SYSTEM sorting_by_height_basic
  (* Version 1.0, 2022-10-03, AK123957 *)
  APPLICATION sorting_by_height_basicApp
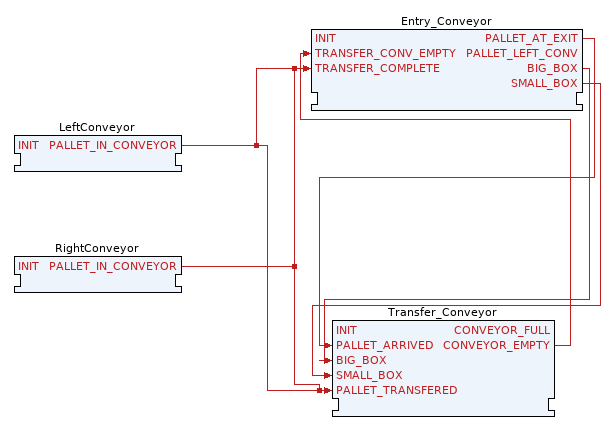
    SUBAPPLICATION Entry_Conveyor
      EVENT_INPUT
        INIT;
        TRANSFER_CONV_EMPTY;
        TRANSFER_COMPLETE;
      END_EVENT
      EVENT_OUTPUT
        PALLET_AT_EXIT;
        PALLET_LEFT_CONV;
        BIG_BOX;
        SMALL_BOX;
      END_EVENT
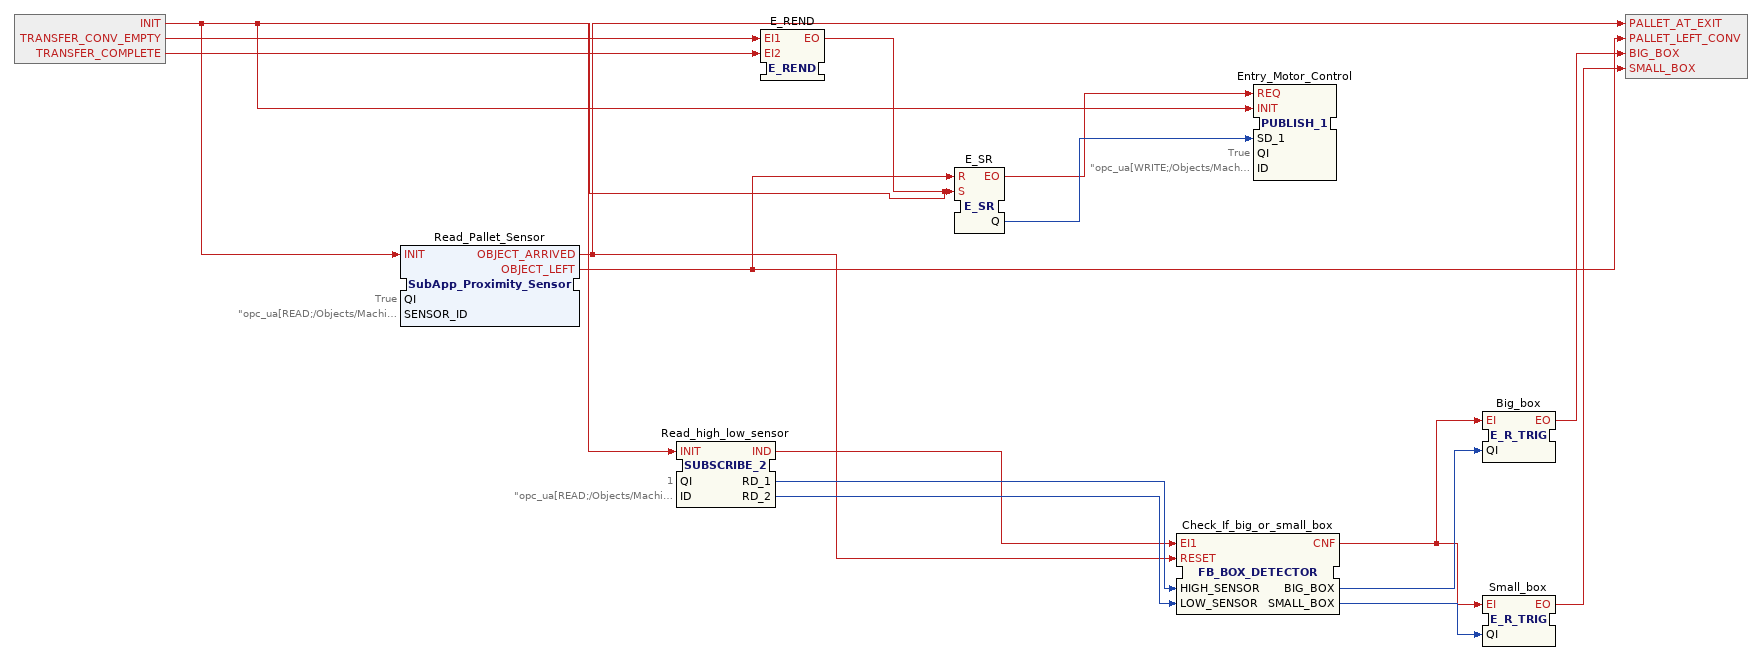
      FBS
        Entry_Motor_Control : PUBLISH_1(QI := True, ID := "opc_ua[WRITE;/Objects/Machines/EntryConveyor/FIO_oEntryMotor,1:s=FIO_oEntryMotor]");
        E_SR : E_SR;
        Check_If_big_or_small_box : FB_BOX_DETECTOR;
        Read_high_low_sensor : SUBSCRIBE_2(QI := 1, ID := "opc_ua[READ;/Objects/Machines/EntryConveyor/FIO_iHighSensor,1:s=FIO_iHighSensor;/Objects/Machines/EntryConveyor/FIO_iLowSensor,1:s=FIO_iLowSensor]");
        Big_box : E_R_TRIG;
        Small_box : E_R_TRIG;
        E_REND : E_REND;
      END_FBS
      SUBAPPS
        Read_Pallet_Sensor : SubApp_Proximity_Sensor(QI := True, SENSOR_ID := "opc_ua[READ;/Objects/Machines/EntryConveyor/FIO_iPalletSensor,1:s=FIO_iPalletSensor]");
      END_SUBAPPS
      EVENT_CONNECTIONS
        E_SR.EO TO Entry_Motor_Control.REQ;
        Read_Pallet_Sensor.OBJECT_ARRIVED TO PALLET_AT_EXIT;
        Read_Pallet_Sensor.OBJECT_LEFT TO PALLET_LEFT_CONV;
        INIT TO Read_Pallet_Sensor.INIT;
        Read_high_low_sensor.IND TO Check_If_big_or_small_box.EI1;
        Read_Pallet_Sensor.OBJECT_ARRIVED TO Check_If_big_or_small_box.RESET;
        Check_If_big_or_small_box.CNF TO Big_box.EI;
        Check_If_big_or_small_box.CNF TO Small_box.EI;
        Big_box.EO TO BIG_BOX;
        Small_box.EO TO SMALL_BOX;
        INIT TO Read_high_low_sensor.INIT;
        INIT TO Entry_Motor_Control.INIT;
        Read_Pallet_Sensor.OBJECT_LEFT TO E_SR.R;
        TRANSFER_CONV_EMPTY TO E_REND.EI1;
        TRANSFER_COMPLETE TO E_REND.EI2;
        E_REND.EO TO E_SR.S;
        INIT TO E_SR.S;
      END_CONNECTIONS
      DATA_CONNECTIONS
        E_SR.Q TO Entry_Motor_Control.SD_1;
        Read_high_low_sensor.RD_1 TO Check_If_big_or_small_box.HIGH_SENSOR;
        Read_high_low_sensor.RD_2 TO Check_If_big_or_small_box.LOW_SENSOR;
        Check_If_big_or_small_box.BIG_BOX TO Big_box.QI;
        Check_If_big_or_small_box.SMALL_BOX TO Small_box.QI;
      END_CONNECTIONS
    END_SUBAPPLICATION
    SUBAPPLICATION LeftConveyor
      EVENT_INPUT
        INIT;
      END_EVENT
      EVENT_OUTPUT
        PALLET_IN_CONVEYOR;
      END_EVENT
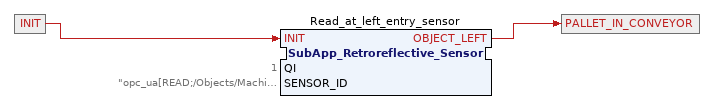
      SUBAPPS
        Read_at_left_entry_sensor : SubApp_Retroreflective_Sensor(QI := 1, SENSOR_ID := "opc_ua[READ;/Objects/Machines/LeftConveyor/FIO_iAtLeftEntry,1:s=FIO_iAtLeftEntry]");
      END_SUBAPPS
      EVENT_CONNECTIONS
        INIT TO Read_at_left_entry_sensor.INIT;
        Read_at_left_entry_sensor.OBJECT_LEFT TO PALLET_IN_CONVEYOR;
      END_CONNECTIONS
    END_SUBAPPLICATION
    SUBAPPLICATION RightConveyor
      EVENT_INPUT
        INIT;
      END_EVENT
      EVENT_OUTPUT
        PALLET_IN_CONVEYOR;
      END_EVENT
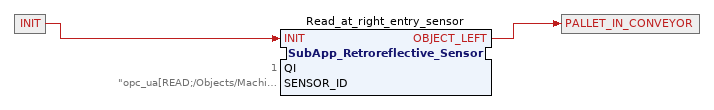
      SUBAPPS
        Read_at_right_entry_sensor : SubApp_Retroreflective_Sensor(QI := 1, SENSOR_ID := "opc_ua[READ;/Objects/Machines/RightConveyor/FIO_iAtRightEntry,1:s=FIO_iAtRightEntry]");
      END_SUBAPPS
      EVENT_CONNECTIONS
        INIT TO Read_at_right_entry_sensor.INIT;
        Read_at_right_entry_sensor.OBJECT_LEFT TO PALLET_IN_CONVEYOR;
      END_CONNECTIONS
    END_SUBAPPLICATION
    SUBAPPLICATION Transfer_Conveyor
      EVENT_INPUT
        INIT;
        PALLET_ARRIVED;
        BIG_BOX;
        SMALL_BOX;
        PALLET_TRANSFERED;
      END_EVENT
      EVENT_OUTPUT
        CONVEYOR_FULL;
        CONVEYOR_EMPTY;
      END_EVENT
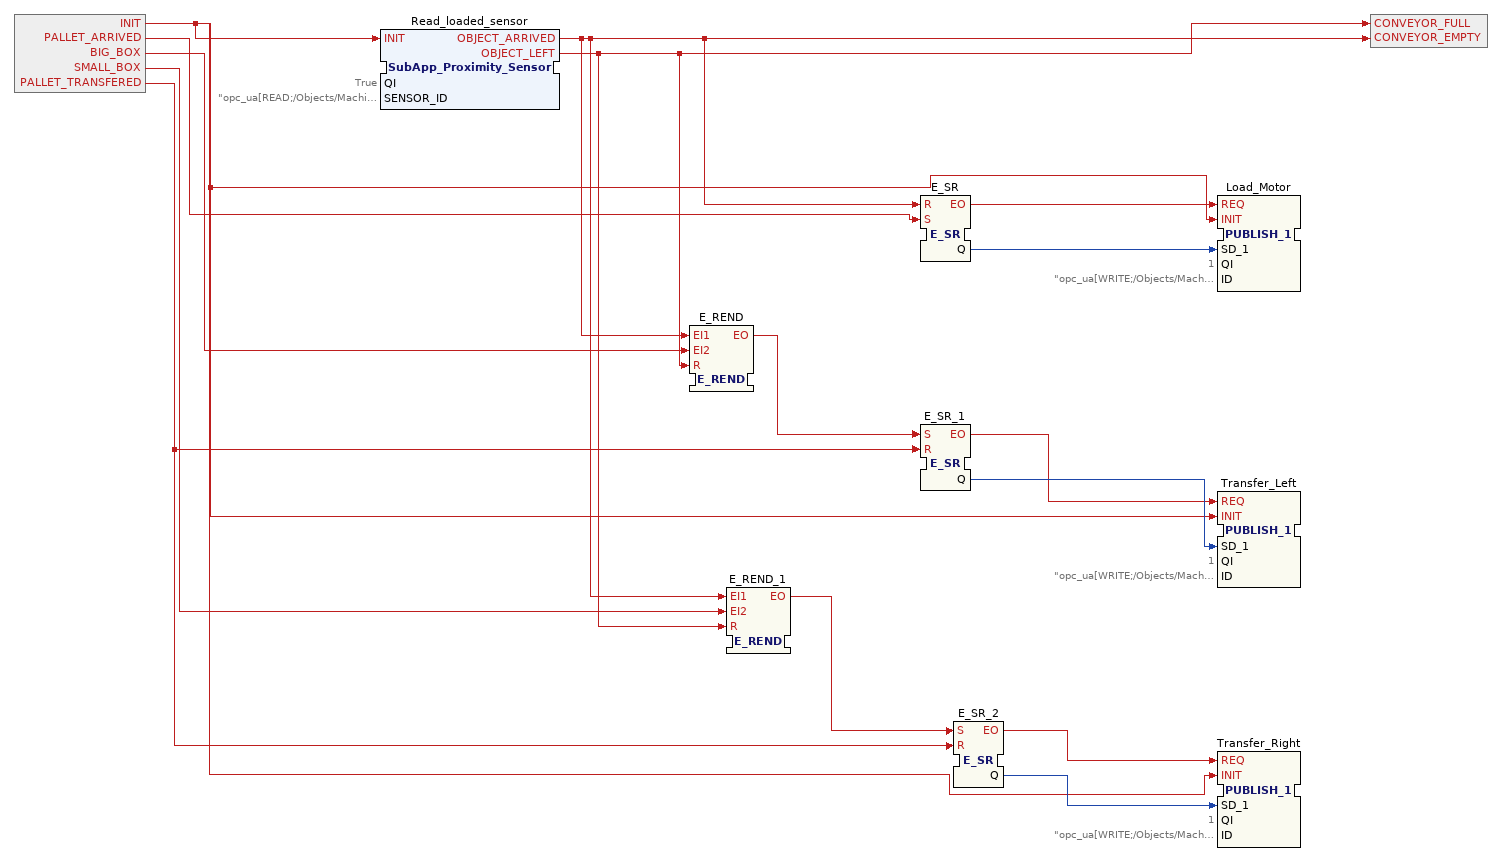
      FBS
        Load_Motor : PUBLISH_1(QI := 1, ID := "opc_ua[WRITE;/Objects/Machines/TransferConveyor/FIO_oLoad,1:s=FIO_oLoad]");
        E_SR : E_SR;
        Transfer_Right : PUBLISH_1(QI := 1, ID := "opc_ua[WRITE;/Objects/Machines/TransferConveyor/FIO_oTransferRight,1:s=FIO_oTransferRight]");
        Transfer_Left : PUBLISH_1(QI := 1, ID := "opc_ua[WRITE;/Objects/Machines/TransferConveyor/FIO_oTransferLeft,1:s=FIO_oTransferLeft]");
        E_REND : E_REND;
        E_SR_1 : E_SR;
        E_SR_2 : E_SR;
        E_REND_1 : E_REND;
      END_FBS
      SUBAPPS
        Read_loaded_sensor : SubApp_Proximity_Sensor(QI := True, SENSOR_ID := "opc_ua[READ;/Objects/Machines/TransferConveyor/FIO_iLoaded,1:s=FIO_iLoaded]");
      END_SUBAPPS
      EVENT_CONNECTIONS
        E_SR.EO TO Load_Motor.REQ;
        E_REND.EO TO E_SR_1.S;
        E_SR_1.EO TO Transfer_Left.REQ;
        E_SR_2.EO TO Transfer_Right.REQ;
        E_REND_1.EO TO E_SR_2.S;
        INIT TO Read_loaded_sensor.INIT;
        Read_loaded_sensor.OBJECT_ARRIVED TO E_SR.R;
        INIT TO Load_Motor.INIT;
        PALLET_ARRIVED TO E_SR.S;
        Read_loaded_sensor.OBJECT_LEFT TO CONVEYOR_EMPTY;
        Read_loaded_sensor.OBJECT_ARRIVED TO CONVEYOR_FULL;
        Read_loaded_sensor.OBJECT_ARRIVED TO E_REND.EI1;
        BIG_BOX TO E_REND.EI2;
        Read_loaded_sensor.OBJECT_ARRIVED TO E_REND_1.EI1;
        SMALL_BOX TO E_REND_1.EI2;
        PALLET_TRANSFERED TO E_SR_1.R;
        PALLET_TRANSFERED TO E_SR_2.R;
        INIT TO Transfer_Left.INIT;
        INIT TO Transfer_Right.INIT;
        Read_loaded_sensor.OBJECT_LEFT TO E_REND.R;
        Read_loaded_sensor.OBJECT_LEFT TO E_REND_1.R;
      END_CONNECTIONS
      DATA_CONNECTIONS
        E_SR.Q TO Load_Motor.SD_1;
        E_SR_1.Q TO Transfer_Left.SD_1;
        E_SR_2.Q TO Transfer_Right.SD_1;
      END_CONNECTIONS
    END_SUBAPPLICATION
    EVENT_CONNECTIONS
      Transfer_Conveyor.CONVEYOR_EMPTY TO Entry_Conveyor.TRANSFER_CONV_EMPTY;
      Entry_Conveyor.PALLET_AT_EXIT TO Transfer_Conveyor.PALLET_ARRIVED;
      Entry_Conveyor.BIG_BOX TO Transfer_Conveyor.BIG_BOX;
      Entry_Conveyor.SMALL_BOX TO Transfer_Conveyor.SMALL_BOX;
      LeftConveyor.PALLET_IN_CONVEYOR TO Entry_Conveyor.TRANSFER_COMPLETE;
      LeftConveyor.PALLET_IN_CONVEYOR TO Transfer_Conveyor.PALLET_TRANSFERED;
      RightConveyor.PALLET_IN_CONVEYOR TO Entry_Conveyor.TRANSFER_COMPLETE;
      RightConveyor.PALLET_IN_CONVEYOR TO Transfer_Conveyor.PALLET_TRANSFERED;
    END_CONNECTIONS
  END_APPLICATION
  DEVICE VM_Ubuntu : FORTE_PC(MGR_ID := "localhost:61499")
    {SET_ATTRIBUTE(Profile, HOLOBLOC)} (* device profile *)
    RESOURCE EMB_RES : EMB_RES
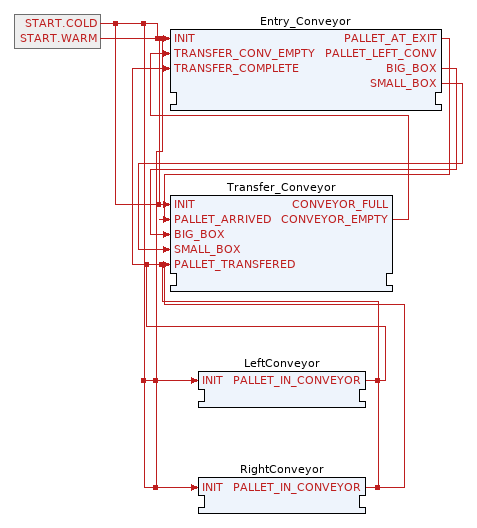
      SUBAPPLICATION Transfer_Conveyor
        EVENT_INPUT
          INIT;
          PALLET_ARRIVED;
          BIG_BOX;
          SMALL_BOX;
          PALLET_TRANSFERED;
        END_EVENT
        EVENT_OUTPUT
          CONVEYOR_FULL;
          CONVEYOR_EMPTY;
        END_EVENT
      END_SUBAPPLICATION
      SUBAPPLICATION Entry_Conveyor
        EVENT_INPUT
          INIT;
          TRANSFER_CONV_EMPTY;
          TRANSFER_COMPLETE;
        END_EVENT
        EVENT_OUTPUT
          PALLET_AT_EXIT;
          PALLET_LEFT_CONV;
          BIG_BOX;
          SMALL_BOX;
        END_EVENT
      END_SUBAPPLICATION
      SUBAPPLICATION RightConveyor
        EVENT_INPUT
          INIT;
        END_EVENT
        EVENT_OUTPUT
          PALLET_IN_CONVEYOR;
        END_EVENT
      END_SUBAPPLICATION
      SUBAPPLICATION LeftConveyor
        EVENT_INPUT
          INIT;
        END_EVENT
        EVENT_OUTPUT
          PALLET_IN_CONVEYOR;
        END_EVENT
      END_SUBAPPLICATION
      EVENT_CONNECTIONS
        START.COLD TO Transfer_Conveyor.INIT;
        START.WARM TO Transfer_Conveyor.INIT;
        Transfer_Conveyor.CONVEYOR_EMPTY TO Entry_Conveyor.TRANSFER_CONV_EMPTY;
        Entry_Conveyor.PALLET_AT_EXIT TO Transfer_Conveyor.PALLET_ARRIVED;
        Entry_Conveyor.BIG_BOX TO Transfer_Conveyor.BIG_BOX;
        Entry_Conveyor.SMALL_BOX TO Transfer_Conveyor.SMALL_BOX;
        START.COLD TO Entry_Conveyor.INIT;
        START.WARM TO Entry_Conveyor.INIT;
        START.COLD TO LeftConveyor.INIT;
        START.COLD TO RightConveyor.INIT;
        START.WARM TO LeftConveyor.INIT;
        START.WARM TO RightConveyor.INIT;
        LeftConveyor.PALLET_IN_CONVEYOR TO Entry_Conveyor.TRANSFER_COMPLETE;
        LeftConveyor.PALLET_IN_CONVEYOR TO Transfer_Conveyor.PALLET_TRANSFERED;
        RightConveyor.PALLET_IN_CONVEYOR TO Entry_Conveyor.TRANSFER_COMPLETE;
        RightConveyor.PALLET_IN_CONVEYOR TO Transfer_Conveyor.PALLET_TRANSFERED;
      END_CONNECTIONS
    END_RESOURCE
  END_DEVICE
  MAPPINGS
    sorting_by_height_basicApp.Transfer_Conveyor ON VM_Ubuntu.EMB_RES.Transfer_Conveyor;
    sorting_by_height_basicApp.Entry_Conveyor ON VM_Ubuntu.EMB_RES.Entry_Conveyor;
    sorting_by_height_basicApp.RightConveyor ON VM_Ubuntu.EMB_RES.RightConveyor;
    sorting_by_height_basicApp.LeftConveyor ON VM_Ubuntu.EMB_RES.LeftConveyor;
  END_MAPPINGS
  SEGMENTS
    Ethernet : Ethernet;
  END_SEGMENTS
  LINKS
    VM_Ubuntu => Ethernet;
  END_LINKS
END_SYSTEM
